TYPE ST_HornLightAr :
STRUCT
    Output      :UINT;
    On          :BOOL;
END_STRUCT
END_TYPE

(* stored: Version 1.1.0.1, ProductVersion 3.1.4020.12
   DUT ST_HornLightAr: Id {0de45d9a-21c3-4079-84d4-a666437f7cc9} *)
